// TIA Portal V20 export
TYPE "LKinCtrl_typeZoneParameters"
   STRUCT
      zoneConfigurationIndex : DInt;   // Index of zone configuration at MovePath
      zoneNumber : DInt;   // Zone number
      deactivationMode : DInt;   // Deactivation mode for zone commands
   END_STRUCT;
END_TYPE
